FUNCTION_BLOCK FB_Axis EXTENDS FB_Device
VAR_INPUT
	Axis				: REFERENCE TO AXIS_REF;
	cmd					: E_AxisCommand := E_AxisCommand.None;
	
	inpPosition			: LREAL;
	inpVelocity			: LREAL := 500.0;
	inpAcceleration		: LREAL := 100.0;
	inpDeceleration		: LREAL := 100.0;
END_VAR
VAR_OUTPUT
	stsState			: E_AxisState := E_AxisState.Off;
	stsFaultCode		: DINT;
	stsPowerOn			: BOOL;
	stsPosition			: LREAL;
	stsVelocity			: LREAL;
END_VAR
VAR
	PowerOn				: MC_Power;
	MoveAbs				: MC_MoveAbsolute;
	MoveVel				: MC_MoveVelocity;
	MoveStop			: MC_Stop;

	PowerOnTimer		: TON;
	StartTimer			: TON;
	StopTimer			: TON;
	PowerOnSimTime		: TIME := T#3S;
	StartSimTime		: TIME := T#3S;
	StopSimTime			: TIME := T#3S;
	PowerOnFailTime		: TIME := T#5S;
	StartFailTime		: TIME := T#5S;
	StopFailTime		: TIME := T#5S;
END_VAR

Map();
Status();
StateMachine();
Control();

METHOD Control : BOOL
VAR_INPUT
END_VAR
IF stsState = E_AxisState.TurningOn THEN
	PowerOn.Enable := TRUE;
	PowerOn.Enable_Negative := TRUE;
	PowerOn.Enable_Positive := TRUE;
END_IF

IF stsState = E_AxisState.TurningOff THEN
	PowerOn.Enable := FALSE;
	PowerOn.Enable_Negative := FALSE;
	PowerOn.Enable_Positive := FALSE;
END_IF

IF stsState = E_AxisState.Stopping THEN
	MoveStop.Execute := TRUE;
END_IF
END_METHOD

METHOD Map : BOOL
VAR_INPUT
END_VAR
MoveAbs(Axis := Axis, Position := inpPosition, Velocity := inpVelocity, Acceleration := inpAcceleration, Deceleration := inpDeceleration);
MoveVel(Axis := Axis, Velocity := inpVelocity, Acceleration := inpAcceleration, Deceleration := inpDeceleration);
MoveStop(Axis := Axis);
PowerOn(Axis := Axis);
END_METHOD

METHOD StateMachine : BOOL
VAR_INPUT
END_VAR
CASE stsState OF
	E_AxisState.Off:
		IF cmd = E_AxisCommand.TurnOn THEN
			stsState := E_AxisState.TurningOn;
		END_IF
	E_AxisState.TurningOn:
		IF stsPowerOn THEN
			stsState := E_AxisState.Ready;
		END_IF
	E_AxisState.Ready:
		IF cmd = E_AxisCommand.ExecuteMoveAbs THEN
			MoveAbs.Execute := TRUE;
		ELSIF cmd = E_AxisCommand.ExecuteMoveVel THEN
			MoveVel.Execute := TRUE;
		ELSIF cmd = E_AxisCommand.Stop THEN
			MoveAbs.Execute := FALSE;
			MoveVel.Execute := FALSE;
			stsState := E_AxisState.Stopping;
		END_IF
		IF MoveAbs.Busy THEN
			MoveAbs.Execute := FALSE;
			MoveVel.Execute := FALSE;
			stsState := E_AxisState.Moving;
		END_IF
	E_AxisState.Moving:
		IF MoveAbs.Done THEN
			stsState := E_AxisState.Ready;
		ELSIF cmd = E_AxisCommand.Stop THEN
			stsState := E_AxisState.Stopping;
		END_IF
	E_AxisState.Stopping:
		IF NOT MoveAbs.Busy THEN
			MoveStop.Execute := FALSE;
			stsState := E_AxisState.Ready;
		END_IF
	E_AxisState.TurningOff:
		IF NOT stsPowerOn THEN
			stsState := E_AxisState.Off;
		END_IF
END_CASE

IF cmd = E_AxisCommand.TurnOff THEN
	stsState := E_AxisState.TurningOff;
END_IF

cmd := E_AxisCommand.None;
END_METHOD

METHOD Status : BOOL
VAR_INPUT
END_VAR
stsPowerOn := PowerOn.Status;
stsPosition := Axis.NcToPlc.ActPos;
stsVelocity := Axis.NcToPlc.ActVelo;
END_METHOD

END_FUNCTION_BLOCK

(* stored: Version 1.1.0.1, ProductVersion 3.1.4024.4
   POU FB_Axis: Id {801782d1-4023-4117-bad0-208e2b5bb926}, SpecialFunc None
   Method Control: Id {5ceeb8c4-6437-404b-91d7-5a4d22eb07ca}
   Method Map: Id {d1aa42fb-74eb-4c00-8dbe-3673a07cccec}
   Method StateMachine: Id {fd7c0724-f298-4847-97d0-6e183c194278}
   Method Status: Id {95f76909-4766-4580-947d-ef2adccc66ce} *)
